{library PUBLIC}
(* Position number type *)
TYPE PositionType : INT(1..9);
END_TYPE

(* stored: Version 1.1.0.1, ProductVersion 3.1.4024.2
   EnumerationTextList PositionType: Id {62c18f4d-7c30-4592-aae5-cbc48d4047c5} *)
